FUNCTION_BLOCK shutdown
VAR_INPUT
	Trig: BOOL;
	Shut: NT_Shutdown;
END_VAR
VAR_OUTPUT
END_VAR
VAR
	Timer: TON;
	Shutd:NT_Shutdown;
END_VAR

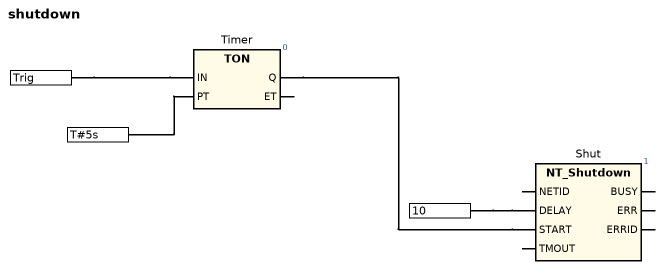
Timer(IN := Trig, PT := T#5s); // TON
Shut(DELAY := 10, START := Timer.Q); // NT_Shutdown

END_FUNCTION_BLOCK

(* stored: Version 1.1.0.1, ProductVersion 3.1.4024.3
   POU shutdown: Id {4266c1c9-f5ca-4158-9adf-7d692743223b}, SpecialFunc None *)
